// TIA Portal project "HochbehaelterDigitalTwin" (V14)

(* hardware
DEVICE "S7-1200-Station_1"  S7-1200 Station
   slot 0: "Baugruppenträger_0"  Rack  V1.0
   slot 1: "PLC"  CPU 1214C DC/DC/DC  6ES7 214-1AG40-0XB0  V4.1
   slot 3: "AQ 1x12BIT_1"  6ES7 232-4HA30-0XB0  V1.0
DEVICE "HMI"  KTP700 Basic PN
   slot 0: "HMI"  HMI  6AV2 123-2GB03-0AX0  13.0.1.0
   slot 1: "HMI_RT_1"  KTP700 Basic PN  6AV2 123-2GB03-0AX0  13.0.1.0
   slot 5: "HMI.IE_CP_1"  PROFINET Schnittstelle
      slot 1: "PROFINET Schnittstelle_1"  PROFINET Schnittstelle
         slot 1: "Port_1"  Port
*)

// ===== PLC "PLC"  CPU 1214C DC/DC/DC =====

VAR_GLOBAL   // PLC tag table "Standard-Variablentabelle"
   "System_Byte" AT %MB100 : Byte;
   "FirstScan" AT %M100.0 : Bool;
   "DiagStatusUpdate" AT %M100.1 : Bool;
   "AlwaysTRUE" AT %M100.2 : Bool;
   "AlwaysFALSE" AT %M100.3 : Bool;
   "Clock_Byte" AT %MB110 : Byte;
   "Clock_10Hz" AT %M110.0 : Bool;
   "Clock_5Hz" AT %M110.1 : Bool;
   "Clock_2.5Hz" AT %M110.2 : Bool;
   "Clock_2Hz" AT %M110.3 : Bool;
   "Clock_1.25Hz" AT %M110.4 : Bool;
   "Clock_1Hz" AT %M110.5 : Bool;
   "Clock_0.625Hz" AT %M110.6 : Bool;
   "Clock_0.5Hz" AT %M110.7 : Bool;
   "Pumpe 1" AT %I0.0 : Bool;
   "Pumpe 2" AT %I0.1 : Bool;
   "Meldeleuchte Pumpe(n)" AT %I0.2 : Bool;
   "Meldeleuchte Motorstörung" AT %I0.3 : Bool;
   "Meldeleuchte Taster Hand" AT %I0.4 : Bool;
   "Meldeleuchte Taster Automatik" AT %I0.5 : Bool;
   "Schwimmerschalter oben" AT %Q0.0 : Bool;
   "Schwimmerschalter unten" AT %Q0.1 : Bool;
   "Schwimmerschalter ganz unten" AT %Q0.2 : Bool;
   "Thermorelais Pumpe 1" AT %Q0.3 : Bool;
   "Thermorelais Pumpe 2" AT %Q0.4 : Bool;
   "Taster Hand" AT %Q0.5 : Bool;
   "Taster Automatik" AT %Q0.6 : Bool;
   "Fuellstand" AT %MW20 : Int;
   "HoherWasserverbrauch" AT %M10.0 : Bool;
   "Pegel" AT %MD40 : Real;
   "Flankenmerker" AT %M0.0 : Bool;
   "Meldeleuchte Hochbehälter leer" AT %I0.6 : Bool;
END_VAR

// folder: System blocks/Program resources

DATA_BLOCK "Taktgeber_100ms"   // DB1
{ S7_Optimized_Access := 'TRUE' }
AUTHOR : Simatic
FAMILY : IEC
NAME : IEC_TMR
VERSION : 1.0
// stored: InstanceOfName IEC_TIMER
"IEC_TIMER"
BEGIN
END_DATA_BLOCK

// folder: (top level)

FUNCTION "fc_HochbehaelterDigitalTwin" : Void   // FC1, SCL
{ S7_Optimized_Access := 'TRUE' }
VERSION : 0.1
BEGIN
   "Taktgeber_100ms".TON(IN:=NOT "Flankenmerker",
                         PT:=t#100ms,
                         Q=>"Flankenmerker");

   IF "Flankenmerker"
   THEN
       // 100ms abgelaufen --> damit die Pegelanzeige nicht so stark springt
       // Der Pegel geht von 0 ... 1000

       IF "Pumpe 1" THEN
           "Pegel" := "Pegel" + 5; // Pumpe 1: Pegel steigt um 5% pro Sekunde
       END_IF;

       IF "Pumpe 2" THEN
           "Pegel" := "Pegel" + 5; // Pumpe 2: Pegel steigt um 5% pro Sekunde
       END_IF;

       "Pegel" := "Pegel" - 1; // Füllstand sinkt durch normalen Verbrauch um 1% pro Sekunde

       IF "HoherWasserverbrauch" THEN
           "Pegel" := "Pegel" - 20; // Füllstand sinkt durch hohem Wasserverbrauch um 20% pro Sekunde
       END_IF;

   END_IF;

   IF "Pegel" > 1000 THEN
       "Pegel" := 1000;    // Pegel nach oben auf 1000 begrenzen
   END_IF;

   IF "Pegel" < 0 THEN
       "Pegel" := 0;// Pegel kann nicht negativ sein
   END_IF;

   "Fuellstand" := "Pegel" / 10;   // Umrechnen von Promille (0..1000) auf Prozent (0..100)

   IF "Fuellstand" > 10 THEN
       "Schwimmerschalter ganz unten" := TRUE;
   ELSE
       "Schwimmerschalter ganz unten" := FALSE;
   END_IF;

   IF "Fuellstand" > 20 THEN
       "Schwimmerschalter unten" := TRUE;
   ELSE
       "Schwimmerschalter unten" := FALSE;
   END_IF;

   IF "Fuellstand" > 90 THEN
       "Schwimmerschalter oben" := TRUE;
   ELSE
       "Schwimmerschalter oben" := FALSE;
   END_IF;
END_FUNCTION

ORGANIZATION_BLOCK "Main"   // OB1, LAD, ProgramCycle
TITLE = "Main Program Sweep (Cycle)"
{ S7_Optimized_Access := 'TRUE' }
VERSION : 0.1
   VAR_INPUT
      Initial_Call : Bool;   // Initial call of this OB
      Remanence : Bool;   // =True, if remanent data are available
   END_VAR
BEGIN

REGION Network 1: -Q1
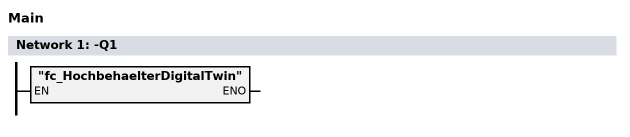
   RUNG wire#powerrail
      "fc_HochbehaelterDigitalTwin"()
   END_RUNG
   // the same network as SCL:
   "fc_HochbehaelterDigitalTwin"();
END_REGION
END_ORGANIZATION_BLOCK

(* ===== HMI "HMI_RT_1" =====
system functions are stored by id; their names below are inferred from use
connection "HMI_Verbindung_1": ETHERNET, SMART_S7_1200_OMS

HMI tags "Standard-Variablentabelle"
   "Fuellstand" : Int = PLC Fuellstand AT %MW20, 100 ms
   "Taster Hand" : Bool = PLC "Taster Hand" AT %Q0.5, 100 ms
   "Meldeleuchte Taster Hand" : Bool = PLC "Meldeleuchte Taster Hand" AT %I0.4, 100 ms
   "Taster Automatik" : Bool = PLC "Taster Automatik" AT %Q0.6, 100 ms
   "Meldeleuchte Taster Automatik" : Bool = PLC "Meldeleuchte Taster Automatik" AT %I0.5, 100 ms
   "Thermorelais Pumpe 1" : Bool = PLC "Thermorelais Pumpe 1" AT %Q0.3, 100 ms
   "Thermorelais Pumpe 2" : Bool = PLC "Thermorelais Pumpe 2" AT %Q0.4, 100 ms
   "Pumpe 1" : Bool = PLC "Pumpe 1" AT %I0.0, 100 ms
   "Pumpe 2" : Bool = PLC "Pumpe 2" AT %I0.1, 100 ms
   "HoherWasserverbrauch" : Bool = PLC HoherWasserverbrauch AT %M10.0, 100 ms
   "MeldeleuchteMotorstoerung" : Bool = PLC "Meldeleuchte Motorstörung" AT %I0.3, 100 ms
   "Meldeleuchte Hochbehälter leer" : Bool = PLC "Meldeleuchte Hochbehälter leer" AT %I0.6, 100 ms
   "Meldeleuchte Pumpe(n)" : Bool = PLC "Meldeleuchte Pumpe(n)" AT %I0.2, 100 ms

screen "HochbehaelterDigitalTwin" 800x480
   TextField "Textfeld_2" at 197,4 size 445x43; Text 'Hochbehälter - Digital Twin'
   Bar "Balken_1" at 91,143 size 136x337; MinimumValue 0; MaximumValue 100
      ProcessValue <- "Fuellstand"
   Button "Schaltfläche_1" at 543,75 size 100x50; TextOff 'Hand'
      on Press: SetBit("Taster Hand")
      on Release: ResetBit("Taster Hand")
      Appearance <- "Meldeleuchte Taster Hand"
   Button "Schaltfläche_2" at 667,75 size 100x50; TextOn 'Automatik'; TextOff 'Automatik'
      on Release: ResetBit("Taster Automatik")
      on Press: SetBit("Taster Automatik")
      Appearance <- "Meldeleuchte Taster Automatik"
   Button "Schaltfläche_4" at 543,420 size 100x50; TextOn 'Thermo 1'; TextOff 'Thermo 1'
      Appearance <- "Thermorelais Pumpe 1"
      on Click: InvertBit("Thermorelais Pumpe 1")
   Button "Schaltfläche_5" at 666,420 size 100x50; TextOn 'Thermo 2'; TextOff 'Thermo 2'
      Appearance <- "Thermorelais Pumpe 2"
      on Click: InvertBit("Thermorelais Pumpe 2")
   Circle "Kreis_1" at 80,56 size 80x80
      Appearance <- "Pumpe 1"
   TextField "Textfeld_1" at 82,84 size 81x23; Text 'Pumpe 1'
   Circle "Kreis_2" at 161,57 size 80x80
      Appearance <- "Pumpe 2"
   TextField "Textfeld_3" at 163,86 size 76x23; Text 'Pumpe 2'
   GraphicView "Oben_Offen" at 250,150 size 60x50; Picture "HMI_Symbole_Schwimmerschalter_Schliesser"
      Visibility <- "Fuellstand"
   GraphicView "Oben_Geschlossen" at 250,150 size 80x50; Picture "HMI_Symbole_Schwimmerschalter_Schliesser_Betaetigt"
      Visibility <- "Fuellstand"
   GraphicView "Mitte_Offen" at 250,350 size 60x50; Picture "HMI_Symbole_Schwimmerschalter_Schliesser"
      Visibility <- "Fuellstand"
   GraphicView "Mitte_Geschlossen" at 250,350 size 80x50; Picture "HMI_Symbole_Schwimmerschalter_Schliesser_Betaetigt"
      Visibility <- "Fuellstand"
   GraphicView "Unten_Offen" at 250,420 size 60x50; Picture "HMI_Symbole_Schwimmerschalter_Schliesser"
      Visibility <- "Fuellstand"
   GraphicView "Unten_Geschlossen" at 250,420 size 80x50; Picture "HMI_Symbole_Schwimmerschalter_Schliesser_Betaetigt"
      Visibility <- "Fuellstand"
   Button "Schaltfläche_6" at 541,351 size 225x50; TextOff 'Hoher Wasserverbrauch'
      on Click: InvertBit("HoherWasserverbrauch")
      Appearance <- "HoherWasserverbrauch"
   Circle "Kreis_3" at 540,197 size 60x60
      Appearance <- "MeldeleuchteMotorstoerung"
   TextField "Textfeld_4" at 600,205 size 120x42; Text 'Motorstörung Pumpe 1 / 2'
   Circle "Kreis_4" at 540,256 size 60x60
      Appearance <- "Meldeleuchte Hochbehälter leer"
   TextField "Textfeld_5" at 600,275 size 151x23; Text 'Hochbehälter leer'
   Circle "Kreis_5" at 540,138 size 60x60
      Appearance <- "Meldeleuchte Pumpe(n)"
   TextField "Textfeld_6" at 600,154 size 115x23; Text 'Pumpe(n) Ein'
*)